// TIA Portal V18 export
VAR_GLOBAL   // PLC tag table "Level"
   Floater_Switch_01 AT %I8.7 : Bool;
   Floater_Switch_02 AT %I9.0 : Bool;
   Floater_Switch_03 AT %I9.1 : Bool;
   Floater_Switch_04 AT %I9.2 : Bool;
   Floater_Switch_05 AT %I9.3 : Bool;
   Floater_Switch_06 AT %I9.4 : Bool;
   Floater_Switch_07 AT %I9.5 : Bool;
   Floater_Switch_08 AT %I9.6 : Bool;
   Floater_Switch_09 AT %I9.7 : Bool;
END_VAR
